{attribute 'reflection'} 
FUNCTION_BLOCK FB_System
VAR_INPUT
	fbAdsMessageHandler 	: FB_AdsMessageHandler;
	fbRecordData 			: FB_RecordData(refAdsMessageHandler := fbAdsMessageHandler);
END_VAR

VAR
	Control				AT %Q* : BYTE; //{simulation-interface}
	Status				AT %I* : BYTE; //{simulation-interface}
	TimeScaling			AT %I* : REAL := 1.0; //{simulation-interface}
	
	{attribute 'instance-path'} 
    {attribute 'noinit'} 
	_sPath 				: STRING;
	
	_bDebug				: BOOL;
	_bVerbose			: BOOL;
	_fDeltaTime 		: REAL;
	_fTimeScaling 		: REAL;
	_eControllerType	: E_ControllerType;
	
	fbPing				: FB_Ping;
	
	{attribute 'hide'}
	fbGetCurTaskIdx 	: TC2_SYSTEM.GETCURTASKINDEX;
END_VAR

InitRun();
fTimeScaling := TimeScaling;
fbPing(bFeedback := Status.7, bTrigger => Control.7);

fbRecordData(); //Execution order -1 relative to FB_AdsMessageHandler
fbAdsMessageHandler();

PROPERTY PUBLIC fTimeScaling : REAL
SET
IF fTimeScaling = 0 THEN
	_fTimeScaling := 1.0;
ELSE
	_fTimeScaling := LIMIT(0.01000001, fTimeScaling, 100.0);	
END_IF
END_SET
GET
fTimeScaling := _fTimeScaling;
END_GET
END_PROPERTY

PROPERTY eControllerType : E_ControllerType
GET
eControllerType := _eControllerType;
END_GET
SET
_eControllerType := eControllerType;
END_SET
END_PROPERTY

METHOD PRIVATE InitRun
VAR_INST
	bInitRun 			: BOOL := TRUE;
	sMessageFormat   	: T_MAXSTRING := '%s %s';
	sMessage  			: T_MAXSTRING;
	fbFormatString 		: FB_FormatString;
END_VAR
IF NOT bInitRun THEN RETURN; END_IF
bInitRun := FALSE;

IF __ISVALIDREF(GVL_Core.refSystem) THEN	
	fbFormatString(sFormat := sMessageFormat, arg1 := F_STRINGEx(_sPath), arg2 := F_STRINGEx('FB_System has no single instance! Check the PROGRAM declaration'), sOut => sMessage);
	ADSLOGSTR(msgCtrlMask := ADSLOG_MSGTYPE_ERROR, '%s', sMessage);	
ELSE 
	GVL_Core.refSystem REF= THIS^;
END_IF

fbGetCurTaskIdx();
_fDeltaTime := UDINT_TO_REAL(TwinCAT_SystemInfoVarList._TaskInfo[fbGetCurTaskIdx.index].CycleTime / 10000) / 1000.0;
_fTimeScaling := 1;

fbRecordData.eControllerType := _eControllerType;
END_METHOD

PROPERTY PUBLIC fDeltaTime : REAL
SET // PRIVATE
_fDeltaTime := fDeltaTime;
END_SET
GET
fDeltaTime := _fDeltaTime;
END_GET
END_PROPERTY

PROPERTY bDebug : BOOL
GET
bDebug := _bDebug;
END_GET
SET
_bDebug := bDebug;
END_SET
END_PROPERTY

PROPERTY bVerbose : BOOL
GET
bVerbose := _bVerbose;
END_GET
SET
_bVerbose := bVerbose;
END_SET
END_PROPERTY

END_FUNCTION_BLOCK

(* stored: Version 1.1.0.1, ProductVersion 3.1.4024.12
   POU FB_System: Id {be746857-6a84-0550-15a8-342a3cf285ce}, SpecialFunc None
   Property fTimeScaling: Id {24281261-b190-0005-28ac-ab20602e18f0}
   Set Set: Id {d4c9598d-134a-0bed-23ef-a2d8f4ecae49}
   Get Get: Id {faee38d2-3304-0e88-0f7b-41af5f8820f8}
   Property eControllerType: Id {842c1e11-fb2e-020a-0bf0-8814ea6d44dc}
   Get Get: Id {195627f8-584e-0b43-3938-6aac17021e11}
   Set Set: Id {6055c751-a3c8-0dde-2598-286cc2bf75aa}
   Method InitRun: Id {9d176150-042b-075c-25f7-3cdd017d1802}
   Property fDeltaTime: Id {a582fa69-51ab-06a9-395c-44350810ecf2}
   Set Set: Id {0918670c-f79e-015c-1fcf-e67f242830f0}
   Get Get: Id {c39c953f-9cc6-0fa1-0ee4-854ccc5e9713}
   Property bDebug: Id {cb9654c8-3a3b-0513-048d-f0f7e81d2e5a}
   Get Get: Id {3f107974-862f-0a37-2e0d-9a39a4576d72}
   Set Set: Id {4e429cb4-7dba-0d6b-2b19-2a9e7bc9c825}
   Property bVerbose: Id {e8e1e559-0690-046a-0b91-1acb33eba34e}
   Get Get: Id {15cd554f-d71d-0a7e-158c-7c7124160153}
   Set Set: Id {69a98c50-13a5-0296-2433-dfd65361c8ab} *)
